Staubli VAL3: oGripCmd.pgx

public program oGripCmd(num nState (dimensions=1))
begin
  dioSet(oGripCmd,nState)
end
